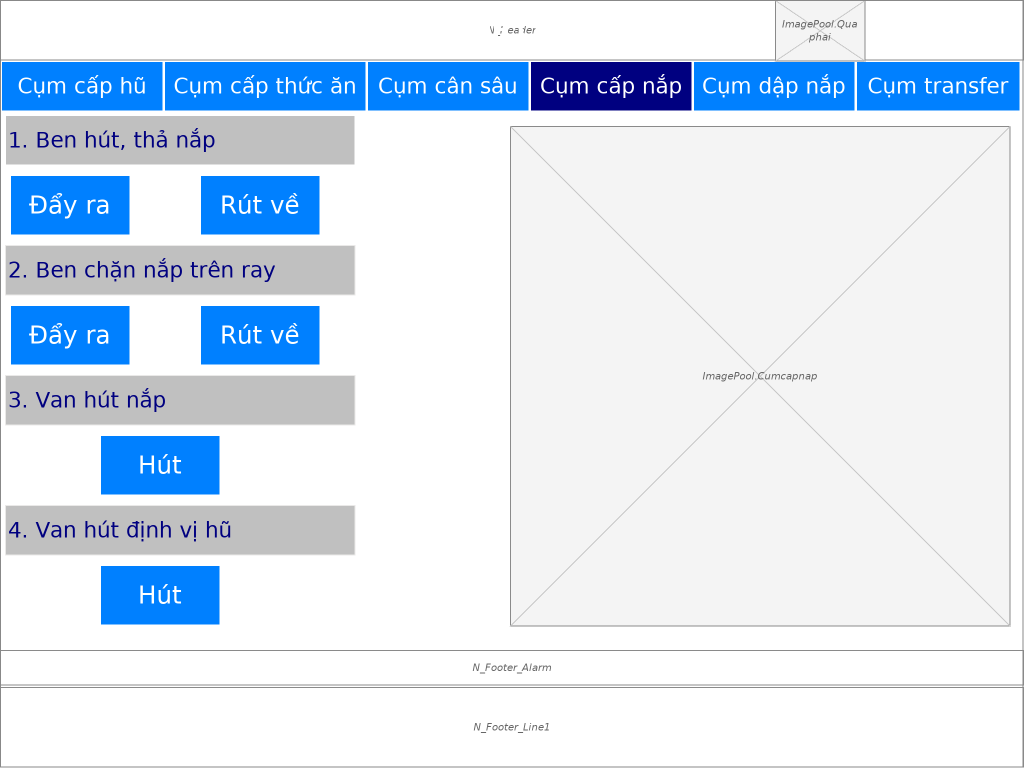
VISUALIZATION N_LidSupply1  // 1024x768
    Rectangle (100,565 120x60), "Dừng hút", invisible if: NOT PR_Line01.bCupSuctionValve, input disabled if: NOT PR_Line01.bCupSuctionValve
        OnMouseDown: execute { PR_Line01.bCupSuctionValve := false; }
    Rectangle (100,435 120x60), "Dừng hút", invisible if: not PR_Line01.bLidSuctionValve, input disabled if: not PR_Line01.bLidSuctionValve
        OnMouseDown: execute { PR_Line01.bLidSuctionValve := FALSE; }
    Rectangle (10,305 120x60), "Đẩy ra", colour toggle: PR_Line01.bCylinder_LidStopper_extend
        OnMouseDown: execute { PR_Line01.bCylinder_LidStopper_extend := TRUE; PR_Line01.bCylinder_LidStopper_retract := FALSE; }
    Rectangle (10,175 120x60), "Đẩy ra", colour toggle: PR_Line01.bCylinder_Suction_extend
        OnMouseDown: execute { PR_Line01.bCylinder_Suction_extend := TRUE; PR_Line01.bCylinder_Suction_retract := FALSE; }
    Rectangle (200,305 120x60), "Rút về", colour toggle: PR_Line01.bCylinder_LidStopper_retract
        OnMouseDown: execute { PR_Line01.bCylinder_LidStopper_retract := TRUE; PR_Line01.bCylinder_LidStopper_extend := FALSE; }
    Frame (0,687 1024x80)
        shows N_Footer_Line1()
    Frame (0,0 1024x60)
        shows N_Header()
    Textfield (353,5 400x50), "MÀN HÌNH CHẠY TAY LINE 1"
    Rectangle (5,115 350x50), "1. Ben hút, thả nắp"
    Rectangle (200,175 120x60), "Rút về", colour toggle: PR_Line01.bCylinder_Suction_retract
        toggle GVL_OF_VU.bValveBlowLid[1]
        OnMouseDown: execute { PR_Line01.bCylinder_Suction_retract := TRUE; PR_Line01.bCylinder_Suction_extend := FALSE; }
    Rectangle (5,245 350x50), "2. Ben chặn nắp trên ray"
    Rectangle (1,61 162x50), "Cụm cấp hũ"
        OnMouseClick: change screen: N_JarSupply1
    Rectangle (164,61 202x50), "Cụm cấp thức ăn"
        OnMouseClick: change screen: N_FoodSupply1
    Rectangle (367,61 162x50), "Cụm cân sâu"
        OnMouseClick: change screen: N_WormWeight1
    Rectangle (530,61 162x50), "Cụm cấp nắp"
        OnMouseClick: change screen: N_LidSupply1
    Rectangle (693,61 162x50), "Cụm dập nắp"
        OnMouseClick: change screen: N_LidPressing1
    Rectangle (856,61 164x50), "Cụm transfer"
        OnMouseClick: change screen: N_Tranfer1
    Rectangle (5,375 350x50), "3. Van hút nắp"
    Rectangle (100,435 120x60), "Hút", invisible if: PR_Line01.bLidSuctionValve, input disabled if: PR_Line01.bLidSuctionValve
        OnMouseDown: execute { PR_Line01.bLidSuctionValve := TRUE; }
    Image (775,0 90x61), input disabled if: bResetAuto2, image: ImagePool.Qua phai
        OnMouseClick: change screen: N_LidSupply2
        OnMouseClick: execute { MAIN_LINE2.bModeManual := TRUE; MAIN_LINE2.bModeAuto := FALSE; }
    Rectangle (5,505 350x50), "4. Van hút định vị hũ"
    Rectangle (100,565 120x60), "Hút", invisible if: PR_Line01.bCupSuctionValve, input disabled if: PR_Line01.bCupSuctionValve
        OnMouseDown: execute { PR_Line01.bCupSuctionValve := true; }
    Image (510,126 500x500), image: ImagePool.Cumcapnap
    Frame (0,650 1024x35)
        shows N_Footer_Alarm()
END_VISUALIZATION

(* stored: Version 1.1.0.1, ProductVersion 3.1.4024.12
   Visu N_LidSupply1: Id {822fb873-d591-4f05-8347-08c7cdc761fe} *)
